// TIA Portal project "PC System" (V14)

(* hardware
DEVICE "S7-1200 station_1"  S7-1200 Station
   slot 0: "Rack_0"  S7-1200 Rack  Rack  V1.0
   slot 1: "Controller"  CPU 1214C DC/DC/DC  6ES7 214-1AG40-0XB0  V4.2
DEVICE "Limon_PC"  SIMATIC PC station
   slot 0: "SIMATIC PC station"  Rail  SIMATIC PC-Station  V1.0
      slot 125: "Stationmanager"  Station_Manager  V6.0.4
   slot 1: "HMI_RT_1"  WinCC RT Advanced  6AV2 104-0xxxx-xxxx  14.0.1.0
      slot 33792: "Host interface"  Host interface
   slot 2: "IE general_1"  IE General  IE_CP  V8.2.0
*)

// ===== PLC "Controller"  CPU 1214C DC/DC/DC =====

VAR_GLOBAL   // PLC tag table "Default tag table"
   "start" AT %I0.0 : Bool;
   "stop" AT %I0.1 : Bool;
   "L1" AT %Q0.1 : Bool;
   "start_hmi" AT %M2.0 : Bool;
   "stop_hmi" AT %M2.1 : Bool;
END_VAR

FUNCTION "AP_HMI" : Void   // FC1, LAD
{ S7_Optimized_Access := 'TRUE' }
VERSION : 0.1
BEGIN

REGION Network 1
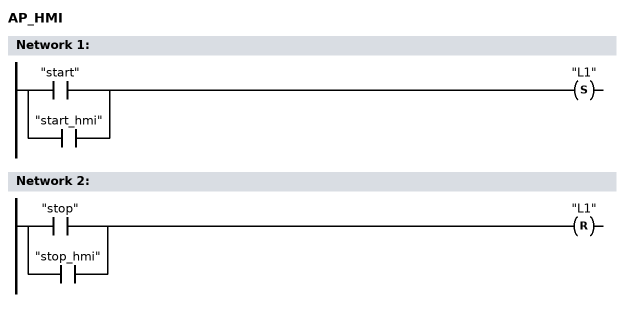
   RUNG wire#powerrail
      Contact( "start" )
      wire#w1
      S_Coil( "L1" )
   END_RUNG
   RUNG wire#powerrail
      Contact( "start_hmi" )
   END_RUNG wire#w1
   // the same network as SCL:
   IF "start" OR "start_hmi" THEN "L1" := TRUE; END_IF;
END_REGION

REGION Network 2
   RUNG wire#powerrail
      Contact( "stop" )
      wire#w1
      R_Coil( "L1" )
   END_RUNG
   RUNG wire#powerrail
      Contact( "stop_hmi" )
   END_RUNG wire#w1
   // the same network as SCL:
   IF "stop" OR "stop_hmi" THEN "L1" := FALSE; END_IF;
END_REGION
END_FUNCTION

ORGANIZATION_BLOCK "Main"   // OB1, LAD, ProgramCycle
TITLE = "Main Program Sweep (Cycle)"
{ S7_Optimized_Access := 'TRUE' }
VERSION : 0.1
   VAR_INPUT
      Initial_Call : Bool;   // Initial call of this OB
      Remanence : Bool;   // =True, if remanent data are available
   END_VAR
BEGIN

REGION Network 1
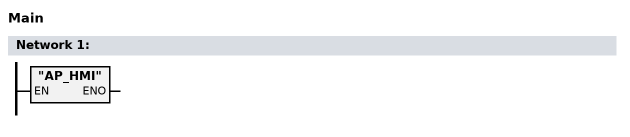
   RUNG wire#powerrail
      "AP_HMI"()
   END_RUNG
   // the same network as SCL:
   "AP_HMI"();
END_REGION
END_ORGANIZATION_BLOCK

(* ===== HMI "HMI_RT_1" =====
system functions are stored by id; their names below are inferred from use
connection "HMI_Connection_1": ETHERNET, S7_1200_OMS

HMI tags "Default tag table"
   "HMI_Tag_1" : Int, internal
   "green_button" : Bool = PLC start_hmi AT %M2.0, 1 s
   "red_button" : Bool = PLC stop_hmi AT %M2.1, 1 s
   "lamp" : Bool = PLC L1 AT %Q0.1, 1 s

Template "Template_1" 800x600
   TextField "Template_Text field_1" at 307,28 size 106x22; Text 'Aplicación PC'

screen "Screen_1" 800x600, template "Template_1"
   Switch "Pushbutton_Round_G" at 145,132 size 50x50; CaptionText 'Switch'; TextOff '0'; TextOn '1'; PictureOff "Pushbutton_Round_G_Off_256c"; PictureOn "Pushbutton_Round_G_On_256c"
      ProcessValue <- "green_button"
   Switch "Pushbutton_Round_R" at 145,237 size 50x50; CaptionText 'Switch'; TextOff '0'; TextOn '1'; PictureOff "Pushbutton_Round_R_Off_256c"; PictureOn "Pushbutton_Round_R_On_256c"
      ProcessValue <- "red_button"
   GraphicIOField "PlotLight_Square_N_Mono" at 369,175 size 50x50; PictureOn "PilotLight_Square_N_On_mono"; PictureOff "PilotLight_Square_N_Off_mono"
      ProcessValue <- "lamp"
   Button "SB_ExitRuntime_85x64" at 616,248 size 85x64; TextOff 'Text'; PictureOff "SB_ExitRuntime_85x64_256c"
      on Click: StopRuntime(0)
*)